# B&R Automation Studio project TestAsProj
Automation Studio 4.12.2.93; Project for testing the OpcUaUnitTesting Python script; technology packages: mappView 5.19.0

## Configuration ARSim

CPU PC_any, AutomationRuntime B4.93, Build 4.1.2, Safety 0.0, Vc 

### Task classes (Cpu.sw)
```
Cyclic#1 (cycle 1000 us, tolerance 0 us):
  BasicTest <- BasicTest.prg
  WaterHeat <- WaterHeat.prg
Cyclic#2 (cycle 10000 us, tolerance 10000 us):
  GetInfo <- GetInfo.prg
Binaries: udbdef, mvLoader, FWRules, OpcUaSrv, TCData, arsvcreg, TCLang, sysconf, Role, User, iomap, ashwd, asfw, arconfig, ashwac, Config_1, TC, Config
Libraries: AsARCfg, runtime, AsBrStr, astime, arssl, fileio, asieccon, aruser, sys_lib, dataobj, standard
```

### Hardware
```
PC : PC_any v1.1.1.0 (OrderNumber=PC)
  ConfigurationID = TestAsProj_ARSim
  SystemTick = 1000
  Cyclic1Duration = 1000
  Cyclic1Tolerance = 0
  Cyclic2Duration = 10000
  Cyclic2Tolerance = 10000
  FileDevice1
  FileDeviceName1 = USER
  FileDevicePath1 = USER_PATH
  FileDevice2
  FileDeviceName2 = FD_Audit
  FileDevicePath2 = C:\BrData\Audit\
  ActivateOpcUa = 1
  OpcUaInformationModels_PV_Version = 1
```

### Config.mpaudittrail - PC/mappServices/Config.mpaudittrail
```
Element gAuditTrail (Type=mpaudittrail)
  Audit:
    Events:
      [0] = 16
      [1] = 19
    TextSource = TXT
      OutputFormat = MpAudit/Event/Root
    Export:
      Encrypt = FALSE
  Alarms = MpAlarmX
```

## Logical view

Binary libraries used (declarations not repeated): operator, runtime, astime, standard, AsIecCon, AsBrStr, AsARCfg

### Global.typ - Global data types
```iecst
(*
OpcUaUnitTesting Example Automation Studio project - Global datatypes

Author: Marcus Mangel (marcus.mangel@br-automation.com)
Date: 27 September 2022
*)
TYPE
	GlobalTestStruct : 	STRUCT  (*Testing using a basic structure*)
		TestUDINT : UDINT; (*Testing with Unsigned Double Integer*)
		TestBOOL : BOOL; (*Testing with Boolean*)
		TestSTRING : STRING[50]; (*Testing with String*)
		TestSubStruct : GlobalTestSubStruct; (*Testing using a structure in a structure (structure-ception)*)
	END_STRUCT;
	GlobalTestSubStruct : 	STRUCT  (*Testing using a structure in a structure (structure-ception)*)
		TestREAL : REAL; (*Testing with REAL*)
		TestLREAL : LREAL; (*Testing with Long REAL*)
	END_STRUCT;
END_TYPE
```

### Global.var - Global variables
```iecst
(*
OpcUaUnitTesting Example Automation Studio project - Global variables

Author: Marcus Mangel (marcus.mangel@br-automation.com)
Date: 27 September 2022
*)
VAR
	gGlobalInt : INT := -100; (*Testing with Integer*)
	gGlobalUInt : UINT := 100; (*Testing with Unsigned Integer*)
	gGlobalString : STRING[50] := 'Test String?!'; (*Testing with String*)
	gTestStruct : GlobalTestStruct := (TestUDINT:=45678,TestBOOL:=TRUE,TestSTRING:='Test String 2',TestSubStruct:=(TestREAL:=123.4,TestLREAL:=432.1)); (*Testing using a basic structure*)
END_VAR
```

### Package Logical/Libraries - Global libraries

- Visualisation Logical/mappView (not shown)

### Program Logical/GetInfo (IEC)

#### Types.typ
```iecst
(*
OpcUaUnitTesting Example Automation Studio project - GetInfo task datatypes

Author: Marcus Mangel (marcus.mangel@br-automation.com)
Date: 27 September 2022
*)

TYPE
	VisInfo_type : 	STRUCT  (*Contains all information shown on the HMI*)
		IpAddr : STRING[80]; (*PLC's IP Address*)
		IsItFriday : STRING[10]; (*String showing the answer to the question "Is it Friday yet?"*)
	END_STRUCT;
	InfoRefreshState_enum :
		( (*State machine states*)
		INFO_REFRESH_STATE_WAIT, (*Wait for a command*)
		INFO_REFRESH_STATE_GET_IP, (*Get the PLC's IP Address*)
		INFO_REFRESH_STATE_GET_DAY, (*Figure out if today is Friday*)
		INFO_REFRESH_STATE_ERROR (*Error refreshing information*)
		);
END_TYPE
```

#### Variables.var
```iecst
(*
OpcUaUnitTesting Example Automation Studio project - GetInfo task variables

Author: Marcus Mangel (marcus.mangel@br-automation.com)
Date: 27 September 2022
*)
VAR
	VisInfo : VisInfo_type; (*Contains all information shown on the HMI*)
	InfoRefreshState : InfoRefreshState_enum; (*State machine state*)
	CmdRefreshInfo : BOOL; (*Command to start refreshing information*)
	CmdErrorReset : BOOL; (*Reset errors*)
	Error : BOOL; (*Error status*)
	DtStruct : DTStructure; (*Current Date/Time found during refresh*)
END_VAR
(*Function Blocks*)
VAR
	fb_CfgGetIpAddr : CfgGetIPAddr; (*Get PLC's IP Address*)
	fb_DTStructureGetTime : DTStructureGetTime; (*Get current Date/Time*)
END_VAR
```

#### Main.st
```iecst
(*
OpcUaUnitTesting Example Automation Studio project - GetInfo task.
This task populates the ContentInfo content of the mappView HMI

Author: Marcus Mangel (marcus.mangel@br-automation.com)
Date: 27 September 2022
*)

PROGRAM _INIT
    CmdRefreshInfo := TRUE; // Refresh all information on startup

END_PROGRAM

PROGRAM _CYCLIC
    // Refresh Info state machine
    CASE InfoRefreshState OF
        INFO_REFRESH_STATE_WAIT: // Wait for a command
            IF CmdRefreshInfo THEN
                CmdRefreshInfo := FALSE;
                InfoRefreshState := INFO_REFRESH_STATE_GET_IP;
            END_IF;

        INFO_REFRESH_STATE_GET_IP: // Get the PLC's IP Address
            fb_CfgGetIpAddr.enable := TRUE;
            fb_CfgGetIpAddr.pDevice := ADR('IF3');
            fb_CfgGetIpAddr.pIPAddr := ADR(VisInfo.IpAddr);
            fb_CfgGetIpAddr.Len := SIZEOF(VisInfo.IpAddr);

            IF (fb_CfgGetIpAddr.status <> ERR_FUB_BUSY) AND (fb_CfgGetIpAddr.status <> ERR_FUB_ENABLE_FALSE) THEN
                IF fb_CfgGetIpAddr.status = ERR_OK THEN
                    fb_CfgGetIpAddr.enable := FALSE;
                    InfoRefreshState := INFO_REFRESH_STATE_GET_DAY;
                ELSE
                    Error := TRUE;
                    InfoRefreshState := INFO_REFRESH_STATE_ERROR;
                END_IF;
            END_IF;

        INFO_REFRESH_STATE_GET_DAY: // Figure out if it's Friday
            brsmemset(ADR(VisInfo.IsItFriday), 0, SIZEOF(VisInfo.IsItFriday));
            brsstrcpy(ADR(VisInfo.IsItFriday), ADR('No :('));

            fb_DTStructureGetTime.enable := TRUE;
            fb_DTStructureGetTime.pDTStructure := ADR(DtStruct);

            IF (fb_DTStructureGetTime.status <> ERR_FUB_BUSY) AND (fb_DTStructureGetTime.status <> ERR_FUB_ENABLE_FALSE) THEN
                IF fb_DTStructureGetTime.status = ERR_OK THEN
                    fb_DTStructureGetTime.enable := FALSE;
                    IF DtStruct.wday = 5 THEN
                        brsmemset(ADR(VisInfo.IsItFriday), 0, SIZEOF(VisInfo.IsItFriday));
                        brsstrcpy(ADR(VisInfo.IsItFriday), ADR('Yes!'));
                    END_IF;
                    InfoRefreshState := INFO_REFRESH_STATE_WAIT;
                ELSE
                    Error := TRUE;
                    InfoRefreshState := INFO_REFRESH_STATE_ERROR;
                END_IF;
            END_IF;

        INFO_REFRESH_STATE_ERROR: // Error getting info
            IF CmdErrorReset THEN
                CmdErrorReset := FALSE;
                Error := FALSE;
                fb_CfgGetIpAddr.enable := FALSE;
                InfoRefreshState := INFO_REFRESH_STATE_WAIT;
            END_IF;

    END_CASE;

    //Call function blocks
    fb_CfgGetIpAddr();
    fb_DTStructureGetTime();
END_PROGRAM
```

### Program Logical/BasicTest (IEC)

#### Variables.var
```iecst
(*
OpcUaUnitTesting Example Automation Studio project - BasicTest task variables

Author: Marcus Mangel (marcus.mangel@br-automation.com)
Date: 27 September 2022
*)
VAR
	TestBOOL : BOOL := TRUE; (*Boolean variable to test with*)
	TestDINT : DINT := 65534; (*Double Integer variable to test with*)
	TestDT : DATE_AND_TIME; (*DateTime variable to test with*)
	TestTIME : TIME := T#1d; (*Time variable to test with*)
	AdditionIn1 : REAL; (*Calculator test: Input 1*)
	AdditionIn2 : REAL; (*Calculator test: Input 2*)
	AdditionOut : REAL; (*Calculator test: Output*)
END_VAR
```

#### Main.st
```iecst
(*
OpcUaUnitTesting Example Automation Studio project - BasicTest task.
This task provides variables for basic testing.

Author: Marcus Mangel (marcus.mangel@br-automation.com)
Date: 27 September 2022
*)

PROGRAM _INIT
    // Use variables in task so that the compiler includes them
    gGlobalInt;
    gGlobalUInt;
    gGlobalString;
    gTestStruct;

    TestBOOL;
    TestDINT;
    TestDT;
    TestTIME;

END_PROGRAM

PROGRAM _CYCLIC
    // Calculator test
	AdditionOut := AdditionIn1 + AdditionIn2;

END_PROGRAM
```

### Program Logical/WaterHeat (IEC)

#### Variables.var
```iecst
(*
OpcUaUnitTesting Example Automation Studio project - WaterHeat task variables

Author: Marcus Mangel (marcus.mangel@br-automation.com)
Date: 27 September 2022
*)
VAR
	WaterLevel : REAL; (*Level of the water in the heater [%]*)
	WaterTemperature : REAL; (*Temperature of the water in the heater [deg C]*)
	HeaterOn : BOOL; (*Heater is ON if TRUE*)
	FillValveOpen : BOOL; (*Fill Valve is OPEN if TRUE*)
	DrainValveOpen : BOOL; (*Drain Valve is OPEN if TRUE*)
	HeatRate : REAL; (*Rate of water temperature rise [deg C/sec]*)
	CoolRate : REAL; (*Rate of water temperature fall [deg C/sec]*)
	FillRate : REAL; (*Rate of fill [%/sec]*)
	DrainRate : REAL; (*Rate of drain [%/sec]*)
END_VAR
(*Constants*)
VAR CONSTANT
	CYCLES_PER_SECOND : REAL := 1000.0; (*PLC cycles per second for this task's task class*)
	BASE_TEMPERATURE : REAL := 20.0; (*Lowest possible water temperature [deg C]*)
	MAX_TEMPERATURE : REAL := 100.0; (*Highest possible water temperature [deg C]*)
	MIN_LEVEL : REAL := 5.0; (*Minimum water level [%]*)
	MAX_LEVEL : REAL := 100.0; (*Maximum water level [%]*)
END_VAR
```

#### Main.st
```iecst
(*
OpcUaUnitTesting Example Automation Studio project - WaterHeat task.
This task mimics a water heater to provide more advanced testing.

Author: Marcus Mangel (marcus.mangel@br-automation.com)
Date: 27 September 2022
*)

PROGRAM _INIT
    // Initial values
    WaterTemperature := BASE_TEMPERATURE;
    WaterLevel := 0.0;

    HeatRate := 1.0;
    CoolRate := 0.5;
    FillRate := 1.0;
    DrainRate := 1.0;

END_PROGRAM

PROGRAM _CYCLIC
    (*
    This task simulates a water heater which can fill with water and drain water.
    The water inside can also be heated, or cooled to the air if the heater is off.

    The water level will never fall below the MIN_LEVEL constant, nor will it fill above
    the MAX_LEVEL constant. Likewise, it will never heat above the MAX_TEMPERATURE constant and
    it won't cool below the BASE_TEMPERATURE constant.

    Turning the heater on will cause the water to heat at HeatRate. Turning off the heater
    will cause it to cool at CoolRate.

    Opening the fill valve will cause the water to fill at FillRate. Opening the drain
    valve will cause the water to drain at DrainRate. If the fill valve and the drain valve
    are both closed, the water level will not change.

    Rates of change are assumed to be "per second". Therefore, the CYCLES_PER_SECOND constant
    must be consistent with this task's task class cycle time.
    *)

	// Heating
    IF HeaterOn THEN
        WaterTemperature := WaterTemperature + (HeatRate/CYCLES_PER_SECOND);
    ELSE
        WaterTemperature := WaterTemperature - (CoolRate/CYCLES_PER_SECOND);
    END_IF;

    IF WaterTemperature > MAX_TEMPERATURE THEN
        WaterTemperature := MAX_TEMPERATURE;
    ELSIF WaterTemperature < BASE_TEMPERATURE THEN
        WaterTemperature := BASE_TEMPERATURE;
    END_IF;

    // Filling and Draining
    IF FillValveOpen THEN
        WaterLevel := WaterLevel + (FillRate/CYCLES_PER_SECOND);
    END_IF;

    IF DrainValveOpen THEN
        WaterLevel := WaterLevel - (DrainRate/CYCLES_PER_SECOND);
    END_IF;

    IF WaterLevel > MAX_LEVEL THEN
        WaterLevel := MAX_LEVEL;
        FillValveOpen := FALSE;
    ELSIF WaterLevel < MIN_LEVEL THEN
        WaterLevel := MIN_LEVEL;
        DrainValveOpen := FALSE;
    END_IF;

END_PROGRAM
```

### Program Logical/Alarms

#### Variables.var
```iecst
VAR
	fb_MpAlarmXCore : MpAlarmXCore;
END_VAR
```

#### Main.st
```iecst
PROGRAM _INIT
    fb_MpAlarmXCore.MpLink := ADR(gAlarmXCore);
    fb_MpAlarmXCore.Enable := TRUE;

END_PROGRAM

PROGRAM _CYCLIC
	fb_MpAlarmXCore();

END_PROGRAM

PROGRAM _EXIT
	fb_MpAlarmXCore(Enable := FALSE);

END_PROGRAM
```

### Program Logical/Audit

#### Variables.var
```iecst
VAR
	fb_MpAuditTrail : MpAuditTrail;
END_VAR
```

#### Main.st
```iecst
PROGRAM _INIT
    fb_MpAuditTrail.MpLink := ADR(gAuditTrail);
    fb_MpAuditTrail.Enable := TRUE;
    fb_MpAuditTrail.DeviceName := ADR('FD_Audit');

END_PROGRAM

PROGRAM _CYCLIC
	fb_MpAuditTrail();

END_PROGRAM

PROGRAM _EXIT
	fb_MpAuditTrail(Enable := FALSE);

END_PROGRAM
```
